TYPE ST_Area_StorageRoom :
STRUCT
	wpRoom				: ST_WP_StorageRoom;
	fbSpotLights		: FB_DigitalOut;
	fbAlarmsensor		: FB_AlarmSensor(sSensorName := 'StorageRoom', bEnableWarning := FALSE);
END_STRUCT
END_TYPE

(* stored: Version 1.1.0.1, ProductVersion 3.1.4024.12
   DUT ST_Area_StorageRoom: Id {18528100-dda7-484b-86d7-5c53194e685f} *)
